// TIA Portal V20 export
// export: Created 2025-12-01T14:56:17.5997302Z, ExportSetting None, DisplayName Totally Integrated Automation Portal, DisplayVersion V20 Update 3, DisplayName TIA Portal Openness, DisplayVersion V20 Update 3, DisplayName TIA Portal Version Control Interface, DisplayVersion V20 Update 3, DisplayName STEP 7 Professional, DisplayVersion V20 Update 3, DisplayName STEP 7 Safety, DisplayVersion V20 Update 2, DisplayName WinCC Basic/Comfort/Advanced, DisplayVersion V20 Update 3, DisplayName WinCC Professional, DisplayVersion V20 Update 3, DisplayName WinCC Unified, DisplayVersion V20 Update 3
TYPE "UDT_ScadaDatosMaquina"
   STRUCT
      Orden_OP1 : Bool;
      Orden_OP2 : Bool;
      Orden_OP3 : Bool;
      Orden_OP4 : Bool;
      Orden_OP5 : Bool;
      Libre_05 : Bool;
      Libre_06 : Bool;
      Libre_07 : Bool;
      Libre_10 : Bool;
      Libre_11 : Bool;
      Libre_12 : Bool;
      Libre_13 : Bool;
      Libre_14 : Bool;
      Libre_15 : Bool;
      Libre_16 : Bool;
      Libre_17 : Bool;
      Libre_20 : Bool;
      Libre_21 : Bool;
      Libre_22 : Bool;
      Libre_23 : Bool;
      Libre_24 : Bool;
      Libre_25 : Bool;
      Libre_26 : Bool;
      Libre_27 : Bool;
      Libre_30 : Bool;
      Libre_31 : Bool;
      Libre_32 : Bool;
      Libre_33 : Bool;
      Libre_34 : Bool;
      Libre_35 : Bool;
      Libre_36 : Bool;
      Libre_37 : Bool;
      Bultos_OP1 : UInt;
      Bultos_OP2 : UInt;
      Bultos_OP3 : UInt;
      Bultos_OP4 : UInt;
      Bultos_OP5 : UInt;
      TMP_Error : Time_Of_Day;
      Arranques_M1 : UInt;
      TMP_Marcha_M1 : Time_Of_Day;
      Arranques_M2 : UInt;
      TMP_Marcha_M2 : Time_Of_Day;
      Arranques_M3 : UInt;
      TMP_Marcha_M3 : Time_Of_Day;
      MemoBultos_OP1 : Bool;
      MemoBultos_OP2 : Bool;
      MemoBultos_OP3 : Bool;
      MemoBultos_OP4 : Bool;
      MemoBultos_OP5 : Bool;
      MemoArranques_M1 : Bool;
      MemoArranques_M2 : Bool;
      MemoArranques_M3 : Bool;
      Libre_370 : Bool;
      Libre_371 : Bool;
      Libre_372 : Bool;
      Libre_373 : Bool;
      Libre_374 : Bool;
      Libre_375 : Bool;
      Libre_376 : Bool;
      Libre_377 : Bool;
   END_STRUCT;
END_TYPE
